{attribute 'linkalways'} 
{attribute 'no_explicit_call' := 'This FB is a CLASS and must be accessed using methods or properties'}
{attribute 'enable_dynamic_creation'}
FUNCTION_BLOCK Node_F_VN_SetAt_LREAL EXTENDS VisionNode
VAR
    fElement : _LREAL(0.0);
    ipContainer : _ITcVnContainer;
    nIndex : _ULINT(0);
    hrPrev : _HRESULT(S_OK);
    hresult : _HRESULT(S_OK);
END_VAR

METHOD PUBLIC  Clone : I_Node
VAR
	pNode : POINTER TO Node_F_VN_SetAt_LREAL;
END_VAR
pNode := __NEW(Node_F_VN_SetAt_LREAL);
Clone := pNode^;
END_METHOD

METHOD FB_init : BOOL
VAR_INPUT
	bInitRetains : BOOL; // if TRUE, the retain variables are initialized (warm start / cold start)
	bInCopyCode : BOOL;  // if TRUE, the instance afterwards gets moved into the copy code (online change)
END_VAR
AddInput('fElement', fElement);
AddInput('ipContainer', ipContainer);
AddInput('nIndex', nIndex);
AddInput('hrPrev', hrPrev);
AddOutput('ipContainer', ipContainer);
AddOutput('hresult',hresult);
END_METHOD

METHOD PROTECTED OnExecute : HRESULT
hresult.Value := F_VN_SetAt_LREAL(
    fElement := fElement.Value,
    ipContainer := ipContainer.Value,
    nIndex := nIndex.Value,
    hrPrev:= hrPrev.Value);
END_METHOD

METHOD PUBLIC PreExecutionCheck
VAR_INPUT
	Check : I_PreExecutionChecks;
END_VAR
Check.IsTrue(ipContainer.IsValid, 'ipContainer must be a valid container');
Check.IsTrue(ipContainer.HasType('CTcVnContainer_Vector_LREAL'), 'ipContainer contains incorrect types');
END_METHOD

END_FUNCTION_BLOCK

(* stored: Version 1.1.0.1, ProductVersion 3.1.4024.13
   POU Node_F_VN_SetAt_LREAL: Id {12f7b6ea-8a2a-4e55-84a8-78edc59b29ad}, SpecialFunc None
   Folder Constructor: Id {2df4aae0-a639-427e-b26f-4fc72d72c716}
   Method Clone: Id {2c0424ef-867c-4b32-bed7-ea8b23de6c49}
   Method FB_init: Id {d057fd7b-e7b3-4405-99ce-c25de51d6dad}
   Method OnExecute: Id {969caa04-052c-4630-861f-89aaaa5f3996}
   Method PreExecutionCheck: Id {7af055e6-9a73-4ed8-b4ce-2efd1d64916e} *)
